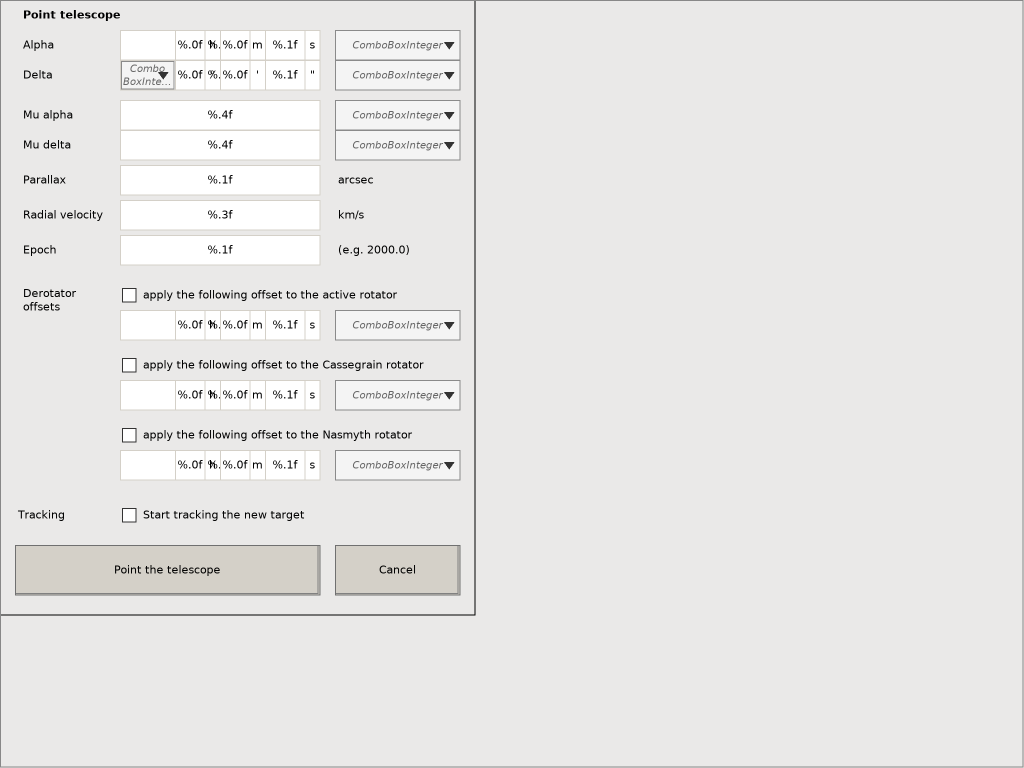
VISUALIZATION VISU_AxesPointDialog  // 1024x768
    Rectangle (0,0 475x615)
    Label (20,5 105x20), "Point telescope"
    Label (20,30 95x30), "Alpha"
    Label (20,60 95x30), "Delta"
    Textfield (120,30 200x30), "%.8f", text variable: GLOBAL.gui.axes.point.field_alpha_decimal, invisible if: GLOBAL.gui.axes.point.units_alpha = AxesDialogAlphaUnits.DIALOG_HMS
        OnMouseClick: write the text variable via VisuDialogs.Numpad
    Textfield (120,60 200x30), "%.8f", text variable: GLOBAL.gui.axes.point.field_delta_decimal, invisible if: GLOBAL.gui.axes.point.units_delta = AxesDialogDeltaUnits.DIALOG_DMS
        OnMouseClick: write the text variable via VisuDialogs.Numpad
    Label (20,100 95x30), "Mu alpha"
    Label (20,130 95x30), "Mu delta"
    Textfield (120,100 200x30), "%.4f", text variable: GLOBAL.gui.axes.point.field_muAlpha
        OnMouseClick: write the text variable via VisuDialogs.Numpad
    Label (20,165 95x30), "Parallax"
    Label (20,200 95x30), "Radial velocity"
    Label (335,200 80x30), "km/s"
    Label (335,165 80x30), "arcsec"
    Textfield (120,130 200x30), "%.4f", text variable: GLOBAL.gui.axes.point.field_muDelta
        OnMouseClick: write the text variable via VisuDialogs.Numpad
    Textfield (120,165 200x30), "%.1f", text variable: GLOBAL.gui.axes.point.field_parallax
        OnMouseClick: write the text variable via VisuDialogs.Numpad
    Textfield (120,200 200x30), "%.3f", text variable: GLOBAL.gui.axes.point.field_radialVelocity
        OnMouseClick: write the text variable via VisuDialogs.Numpad
    Label (20,235 95x30), "Epoch"
    Label (335,235 80x30), "(e.g. 2000.0)"
    Textfield (120,235 200x30), "%.1f", text variable: GLOBAL.gui.axes.point.field_epoch
        OnMouseClick: write the text variable via VisuDialogs.Numpad
    Button (15,545 305x50), "Point the telescope", input disabled if: GLOBAL.mtcs.parts.axes.processes.point.statuses.enabledStatus.disabled
        OnMouseClick: execute { GLOBAL.gui.axes.point.do_request := TRUE; }
        OnMouseClick: CloseDialog Dialog=VISU_AxesPointDialog, Result=OK, NumpadKeypadSet=True
    ComboBoxInteger (335,30 125x30), variable: GLOBAL.gui.axes.point.units_alpha, text list: 'AxesDialogAlphaUnitsTextList'
    ComboBoxInteger (335,60 125x30), variable: GLOBAL.gui.axes.point.units_delta, text list: 'AxesDialogDeltaUnitsTextList'
    ComboBoxInteger (335,100 125x30), variable: GLOBAL.gui.axes.point.units_mu, text list: 'AxesMuUnitsTextList'
    Button (335,545 125x50), "Cancel"
        OnMouseClick: CloseDialog Dialog=VISU_AxesPointDialog, Result=Cancel, NumpadKeypadSet=True
    ComboBoxInteger (335,130 125x30), variable: GLOBAL.gui.axes.point.units_mu, text list: 'AxesMuUnitsTextList'
    Textfield (175,60 30x30), "%.0f", text variable: GLOBAL.gui.axes.point.field_delta_d, invisible if: GLOBAL.gui.axes.point.units_delta <> AxesDialogDeltaUnits.DIALOG_DMS
        OnMouseClick: write the text variable via VisuDialogs.Numpad
    ComboBoxInteger (121,61 53x28), variable: GLOBAL.gui.axes.point.field_delta_sign, invisible if: GLOBAL.gui.axes.point.units_delta <> AxesDialogDeltaUnits.DIALOG_DMS, text list: 'AxesDialogSignTextList'
    Textfield (220,60 30x30), "%.0f", text variable: GLOBAL.gui.axes.point.field_delta_m, invisible if: GLOBAL.gui.axes.point.units_delta <> AxesDialogDeltaUnits.DIALOG_DMS
        OnMouseClick: write the text variable via VisuDialogs.Numpad
    Textfield (265,60 40x30), "%.1f", text variable: GLOBAL.gui.axes.point.field_delta_s, invisible if: GLOBAL.gui.axes.point.units_delta <> AxesDialogDeltaUnits.DIALOG_DMS
        OnMouseClick: write the text variable via VisuDialogs.Numpad
    Label (205,60 15x30), "°", invisible if: GLOBAL.gui.axes.point.units_delta <> AxesDialogDeltaUnits.DIALOG_DMS
    Label (250,60 15x30), "'", invisible if: GLOBAL.gui.axes.point.units_delta <> AxesDialogDeltaUnits.DIALOG_DMS
    Label (305,60 15x30), """, invisible if: GLOBAL.gui.axes.point.units_delta <> AxesDialogDeltaUnits.DIALOG_DMS
    Textfield (175,30 30x30), "%.0f", text variable: GLOBAL.gui.axes.point.field_alpha_h, invisible if: GLOBAL.gui.axes.point.units_alpha <> AxesDialogAlphaUnits.DIALOG_HMS
        OnMouseClick: write the text variable via VisuDialogs.Numpad
    Textfield (220,30 30x30), "%.0f", text variable: GLOBAL.gui.axes.point.field_alpha_m, invisible if: GLOBAL.gui.axes.point.units_alpha <> AxesDialogAlphaUnits.DIALOG_HMS
        OnMouseClick: write the text variable via VisuDialogs.Numpad
    Textfield (265,30 40x30), "%.1f", text variable: GLOBAL.gui.axes.point.field_alpha_s, invisible if: GLOBAL.gui.axes.point.units_alpha <> AxesDialogAlphaUnits.DIALOG_HMS
        OnMouseClick: write the text variable via VisuDialogs.Numpad
    Label (205,30 15x30), "h", invisible if: GLOBAL.gui.axes.point.units_alpha <> AxesDialogAlphaUnits.DIALOG_HMS
    Label (250,30 15x30), "m", invisible if: GLOBAL.gui.axes.point.units_alpha <> AxesDialogAlphaUnits.DIALOG_HMS
    Label (305,30 15x30), "s", invisible if: GLOBAL.gui.axes.point.units_alpha <> AxesDialogAlphaUnits.DIALOG_HMS
    Checkbox (120,500 300x30), "Start tracking the new target", variable: GLOBAL.gui.axes.point.field_tracking
    Label (15,500 95x30), "Tracking"
    Checkbox (120,280 305x30), "apply the following offset to the active rotator", variable: GLOBAL.gui.axes.point.selected_rot, input disabled if: GLOBAL.gui.axes.point.selected_ron OR GLOBAL.gui.axes.point.selected_roc
    Checkbox (120,350 340x30), "apply the following offset to the Cassegrain rotator", variable: GLOBAL.gui.axes.point.selected_roc, input disabled if: GLOBAL.gui.axes.point.selected_rot
    Label (20,280 95x40), "Derotator offsets"
    Textfield (120,310 200x30), "%.8f", text variable: GLOBAL.gui.axes.point.field_rot_decimal, invisible if: GLOBAL.gui.axes.point.units_rot = AxesMoveProcessWidgetUnits.DEGMINSEC, input disabled if: NOT GLOBAL.gui.axes.point.selected_rot
        OnMouseClick: write the text variable via VisuDialogs.Numpad
    ComboBoxInteger (335,310 125x30), variable: GLOBAL.gui.axes.point.units_rot, input disabled if: NOT GLOBAL.gui.axes.point.selected_rot, text list: 'AxesMoveProcessUnitsTextList'
    Textfield (175,310 30x30), "%.0f", text variable: GLOBAL.gui.axes.point.field_rot_d, invisible if: GLOBAL.gui.axes.point.units_rot <> AxesMoveProcessWidgetUnits.DEGMINSEC, input disabled if: NOT GLOBAL.gui.axes.point.selected_rot
        OnMouseClick: write the text variable via VisuDialogs.Numpad
    Textfield (220,310 30x30), "%.0f", text variable: GLOBAL.gui.axes.point.field_rot_m, invisible if: GLOBAL.gui.axes.point.units_rot <> AxesMoveProcessWidgetUnits.DEGMINSEC, input disabled if: NOT GLOBAL.gui.axes.point.selected_rot
        OnMouseClick: write the text variable via VisuDialogs.Numpad
    Textfield (265,310 40x30), "%.1f", text variable: GLOBAL.gui.axes.point.field_rot_s, invisible if: GLOBAL.gui.axes.point.units_rot <> AxesMoveProcessWidgetUnits.DEGMINSEC, input disabled if: NOT GLOBAL.gui.axes.point.selected_rot
        OnMouseClick: write the text variable via VisuDialogs.Numpad
    Label (205,310 15x30), "h", invisible if: GLOBAL.gui.axes.point.units_rot <> AxesMoveProcessWidgetUnits.DEGMINSEC
    Label (250,310 15x30), "m", invisible if: GLOBAL.gui.axes.point.units_rot <> AxesMoveProcessWidgetUnits.DEGMINSEC
    Label (305,310 15x30), "s", invisible if: GLOBAL.gui.axes.point.units_rot <> AxesMoveProcessWidgetUnits.DEGMINSEC
    Checkbox (120,420 335x30), "apply the following offset to the Nasmyth rotator", variable: GLOBAL.gui.axes.point.selected_ron, input disabled if: GLOBAL.gui.axes.point.selected_rot
    Textfield (120,380 200x30), "%.8f", text variable: GLOBAL.gui.axes.point.field_roc_decimal, invisible if: GLOBAL.gui.axes.point.units_rot = AxesMoveProcessWidgetUnits.DEGMINSEC, input disabled if: GLOBAL.gui.axes.point.selected_rot
        OnMouseClick: write the text variable via VisuDialogs.Numpad
    ComboBoxInteger (335,380 125x30), variable: GLOBAL.gui.axes.point.units_rot, input disabled if: GLOBAL.gui.axes.point.selected_rot, text list: 'AxesMoveProcessUnitsTextList'
    Textfield (175,380 30x30), "%.0f", text variable: GLOBAL.gui.axes.point.field_roc_d, invisible if: GLOBAL.gui.axes.point.units_rot <> AxesMoveProcessWidgetUnits.DEGMINSEC, input disabled if: GLOBAL.gui.axes.point.selected_rot
        OnMouseClick: write the text variable via VisuDialogs.Numpad
    Textfield (220,380 30x30), "%.0f", text variable: GLOBAL.gui.axes.point.field_roc_m, invisible if: GLOBAL.gui.axes.point.units_rot <> AxesMoveProcessWidgetUnits.DEGMINSEC, input disabled if: GLOBAL.gui.axes.point.selected_rot
        OnMouseClick: write the text variable via VisuDialogs.Numpad
    Textfield (265,380 40x30), "%.1f", text variable: GLOBAL.gui.axes.point.field_roc_s, invisible if: GLOBAL.gui.axes.point.units_rot <> AxesMoveProcessWidgetUnits.DEGMINSEC, input disabled if: GLOBAL.gui.axes.point.selected_rot
        OnMouseClick: write the text variable via VisuDialogs.Numpad
    Label (205,380 15x30), "h", invisible if: GLOBAL.gui.axes.point.units_rot <> AxesMoveProcessWidgetUnits.DEGMINSEC
    Label (250,380 15x30), "m", invisible if: GLOBAL.gui.axes.point.units_rot <> AxesMoveProcessWidgetUnits.DEGMINSEC
    Label (305,380 15x30), "s", invisible if: GLOBAL.gui.axes.point.units_rot <> AxesMoveProcessWidgetUnits.DEGMINSEC
    Textfield (120,450 200x30), "%.8f", text variable: GLOBAL.gui.axes.point.field_ron_decimal, invisible if: GLOBAL.gui.axes.point.units_rot = AxesMoveProcessWidgetUnits.DEGMINSEC, input disabled if: GLOBAL.gui.axes.point.selected_rot
        OnMouseClick: write the text variable via VisuDialogs.Numpad
    ComboBoxInteger (335,450 125x30), variable: GLOBAL.gui.axes.point.units_rot, input disabled if: GLOBAL.gui.axes.point.selected_rot, text list: 'AxesMoveProcessUnitsTextList'
    Textfield (175,450 30x30), "%.0f", text variable: GLOBAL.gui.axes.point.field_ron_d, invisible if: GLOBAL.gui.axes.point.units_rot <> AxesMoveProcessWidgetUnits.DEGMINSEC, input disabled if: GLOBAL.gui.axes.point.selected_rot
        OnMouseClick: write the text variable via VisuDialogs.Numpad
    Textfield (220,450 30x30), "%.0f", text variable: GLOBAL.gui.axes.point.field_ron_m, invisible if: GLOBAL.gui.axes.point.units_rot <> AxesMoveProcessWidgetUnits.DEGMINSEC, input disabled if: GLOBAL.gui.axes.point.selected_rot
        OnMouseClick: write the text variable via VisuDialogs.Numpad
    Textfield (265,450 40x30), "%.1f", text variable: GLOBAL.gui.axes.point.field_ron_s, invisible if: GLOBAL.gui.axes.point.units_rot <> AxesMoveProcessWidgetUnits.DEGMINSEC, input disabled if: GLOBAL.gui.axes.point.selected_rot
        OnMouseClick: write the text variable via VisuDialogs.Numpad
    Label (205,450 15x30), "h", invisible if: GLOBAL.gui.axes.point.units_rot <> AxesMoveProcessWidgetUnits.DEGMINSEC
    Label (250,450 15x30), "m", invisible if: GLOBAL.gui.axes.point.units_rot <> AxesMoveProcessWidgetUnits.DEGMINSEC
    Label (305,450 15x30), "s", invisible if: GLOBAL.gui.axes.point.units_rot <> AxesMoveProcessWidgetUnits.DEGMINSEC
END_VISUALIZATION

(* stored: Version 1.1.0.1, ProductVersion 3.1.4019.2
   Visu VISU_AxesPointDialog: Id {d8bd5678-9aa9-45df-9243-47a99b604768} *)
